// TIA Portal V20 export
VAR_GLOBAL   // PLC tag table "4.Salida Analoga"
   Output_Analog_1 AT %QW10 : Int;
   Output_Analog_2 AT %QW12 : Int;
   Output_Analog_3 AT %QW14 : Int;
   Output_Analog_4 AT %QW16 : Int;
END_VAR
